TYPE ST_DisplayConfig :
STRUCT
	DisplayName     : STRING(60) := '';  // Vises i HMI
	Description     : STRING(120) := ''; // Detaljeret beskrivelse
	Visible         : BOOL := TRUE;      // Skjul/vis i HMI
	ReadOnly        : BOOL := FALSE;     // Disable write fra HMI
END_STRUCT
END_TYPE

(* stored: Version 1.1.0.1, ProductVersion 3.1.4024.12
   DUT ST_DisplayConfig: Id {12345678-1234-5678-1234-567812345004} *)
